TYPE UDT_DayTime_RD :
STRUCT
times : TIME; // 总时间
timeValue :UDINT; //时间数值
day : USInt; // 天
hour : USInt; // 时
minute : USInt; // 分
second : USInt; // 秒

END_STRUCT
END_TYPE

(* stored: Version 1.1.0.1, ProductVersion 3.1.4024.12
   DUT UDT_DayTime_RD: Id {a554f823-68ea-4b72-9cec-c79cdfac8c26} *)
